// TwinCAT 3 PLC project ReceivingMQTT
// ProgramVersion: 3.1.4022.3
// libraries:
//   Tc2_Standard, * (Beckhoff Automation GmbH)
//   Tc2_System, * (Beckhoff Automation GmbH)
//   Tc3_IotBase, * (Beckhoff Automation GmbH)
//   Tc3_IotCommunicator, * (Beckhoff Automation GmbH)
//   Tc3_JsonXml, * (Beckhoff Automation GmbH)
//   Tc3_Module, * (Beckhoff Automation GmbH)
// project tree:
//   DUTs/ ST_TemperatureStructure.TcDUT
//   GVLs/ Data_Received.TcGVL, Setup_Parameters.TcGVL
//   / PlcTask.TcTTO
//   POUs/ MAIN_Subscriber.TcPOU
// (motion and I/O tree: see PLC project sendingmqtt)
// real-time tasks:
//   TASK PlcTask: cycle T#10ms, priority 20, ADS port 350

CONFIGURATION ReceivingMQTT
    RESOURCE PLC ON TwinCAT3
        TASK PlcTask(INTERVAL := T#10ms, PRIORITY := 20);
        PROGRAM MAIN_Subscriber WITH PlcTask : MAIN_Subscriber;
    END_RESOURCE
END_CONFIGURATION

// ---- DUTs/ST_TemperatureStructure.TcDUT
TYPE ST_TemperatureStructure :
STRUCT
	fRoomTemperature 	: REAL;
	fBathRoomTemperature : REAL;
	diSomeOtherData 		: DINT;
END_STRUCT
END_TYPE

// ---- GVLs/Data_Received.TcGVL
{attribute 'qualified_only'}
VAR_GLOBAL
	stTempData				: ST_TemperatureStructure;	// this is the structured data we will update from the MQTT client
	sJSonStringReceived		: STRING(255);				// this is the latest JSON formatted data string we have recieved
	sPlainStringReceived	: STRING(255);				// this is the latest plain string we have received
	
	// Count the messages sent
	uiJSONReceived				: UINT;
	uiJSONProcessed				: UINT;


	uiPlainReceived				: UINT;

END_VAR

// ---- GVLs/Setup_Parameters.TcGVL
{attribute 'qualified_only'}
VAR_GLOBAL CONSTANT
	sPlainStringTopic	: STRING(255)	:= 'Plain Temperatures';	// this the topic we will publish on for plain string data
	sJsonStringTopic	: STRING(255)	:= 'JSON Temperatures';		// this the topic we will publish on for JSON formatted string data
	sBrokerAddress		: STRING(255)	:= 'test.mosquitto.org';	// this is the address of the MQTT broker we are using
	uiBrokerPort 		: UINT			:= 1883;					// the TCP port for the MQQT broker
END_VAR

// ---- POUs/MAIN_Subscriber.TcPOU
PROGRAM MAIN_Subscriber
VAR
	fbMqttClient		: FB_IotMqttClient;			// The MQTT client for recieving messages
    fbMessageQueue		: FB_IotMqttMessageQueue;	// The message queue for handling recieved messages 
    fbMessage			: FB_IotMqttMessage;		// A message object for processing recieved messages 
	bSubscribed			: BOOL;
	sReceivingTopic		: STRING(255);				// The topic of the last message we recieved 	
	fbJsonDataType 		: FB_JsonReadWriteDataType;	
	fbGetSystemTime		: GETSYSTEMTIME;
	
END_VAR

// Setup the MQTT client (we only do this once when the cods runs for the first time)
fbGetSystemTime();
IF _TaskInfo[GETCURTASKINDEXEX()].FirstCycle THEN    
    fbMqttClient.sHostName      := Setup_Parameters.sBrokerAddress;
    fbMqttClient.nHostPort      := Setup_Parameters.uiBrokerPort;
    fbMqttClient.sTopicPrefix   := '';     
	fbMqttClient.ipMessageQueue := fbMessageQueue;
	fbMqttClient.sClientId 		:= CONCAT('Subscribing_PLC_',DWORD_TO_STRING(fbGetSystemTime.timeLoDW));	// generate and set a psuedorandom client ID 
END_IF

// Run the MQTT client every cycle
fbMqttClient.Execute(bConnect :=true);

IF fbMqttClient.bConnected THEN	// Check that we are connected to the broker 
    IF NOT bSubscribed THEN		// Check if are subscribed, if not we subscribe to the topics of interest to us 

        bSubscribed := fbMqttClient.Subscribe(sTopic:=Setup_Parameters.sPlainStringTopic,
			eQoS:=TcIotMqttQos.AtMostOnceDelivery);
			
        bSubscribed := fbMqttClient.Subscribe(sTopic:=Setup_Parameters.sJsonStringTopic,
			eQoS:=TcIotMqttQos.AtMostOnceDelivery);

    END_IF // check subscription
END_IF // check connection 

// Handle the message queue
IF fbMessageQueue.nQueuedMessages > 0 THEN	// if we have messages in the queue
    IF fbMessageQueue.Dequeue(fbMessage:=fbMessage) THEN	//we pick the latest message, returns TRUE if pick  succeeds
        fbMessage.GetTopic(pTopic:=ADR(sReceivingTopic), nTopicSize:=SIZEOF(sReceivingTopic) );	// get the topic of the message 
		// process the received message based on it's topic 		
		IF sReceivingTopic = Setup_Parameters.sJsonStringTopic THEN	// if the topic is the JSON topic
			IF(fbMessage.GetPayload(pPayload:=ADR(Data_Received.sJSonStringReceived), nPayloadSize:=SIZEOF(Data_Received.sJSonStringReceived), bSetNullTermination:=FALSE)) THEN
				Data_Received.uiJSONReceived	:= Data_Received.uiJSONReceived + 1;	// count JSON messages received
			END_IF // payload retreived
			IF(fbJsonDataType.SetSymbolFromJson(Data_Received.sJSonStringReceived, 'ST_TemperatureStructure', SIZEOF(Data_Received.stTempData), ADR(Data_Received.stTempData))) THEN
				Data_Received.uiJSONProcessed	:= Data_Received.uiJSONProcessed + 1;	// count JSON messages processed
			END_IF // JSON processed 
		ELSIF(sReceivingTopic = Setup_Parameters.sPlainStringTopic) THEN // if the topic is the plain string topic
       		IF(fbMessage.GetPayload(pPayload:=ADR(Data_Received.sPlainStringReceived), nPayloadSize:=SIZEOF(Data_Received.sPlainStringReceived), bSetNullTermination:=FALSE)) THEN
				Data_Received.uiPlainReceived	:= Data_Received.uiPlainReceived + 1;	// count plain messages received
			END_IF	// payload retrieved		
		END_IF // check recieved message topic 
    END_IF // successfully deqeued a message 
END_IF // more than 0 messages in the queue

END_PROGRAM
